PROGRAM general
VAR PERSISTENT
	//System date time function block
	system_date_time : date_time;
	//Daily reset bit, used throughout the program for any resets
	daily_reset : BOOL;
	//Alarm Acknoweldge unlatch timer
	alarm_ack_ton : ton;
	//Alarm Reset unlatch timer
	alarm_reset_ton : ton;
	//Alarm Ack and reset unlatch timer setpoint
	alarm_ack_unlatch_sp : TIME :=T#3S;
	
	safety_reset_ton : TON;
	
	safety_reset AT %Q*  : BOOL;
	safety_error_ack AT %Q* : BOOL;
	safety_run AT %Q*  : BOOL;
	
END_VAR

VAR
	
	safety_reset_ons: R_TRIG;
END_VAR
VAR // added by the converter: edge detectors and wires of the graphical bodies
    _w1 : BOOL;
END_VAR

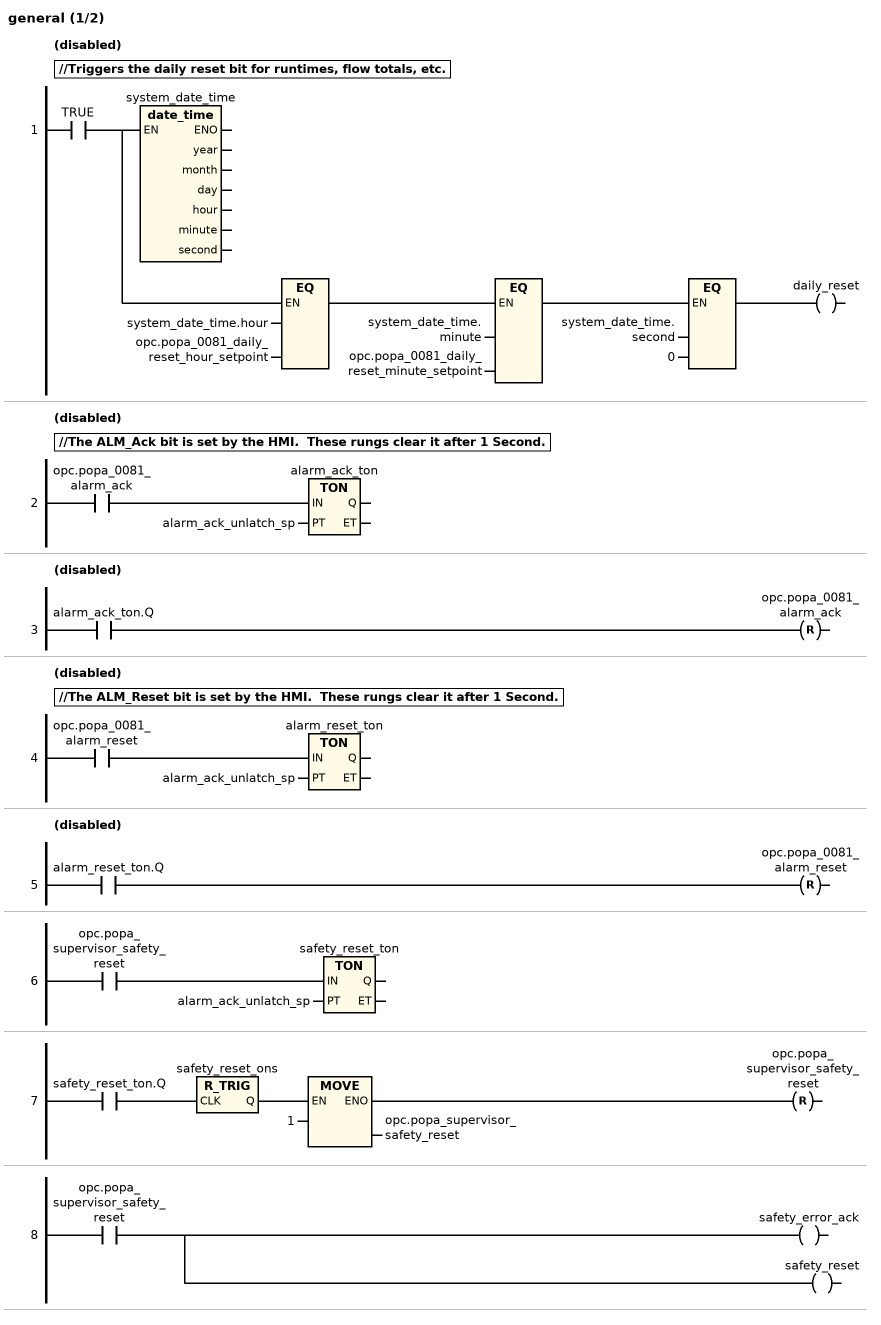
// NETWORK 1 (disabled)
// label: //Triggers the daily reset bit for runtimes, flow totals, etc.
// system_date_time(); // date_time
// daily_reset := system_date_time.hour = opc.popa_0081_daily_reset_hour_setpoint AND system_date_time.minute = opc.popa_0081_daily_reset_minute_setpoint AND system_date_time.second = 0;

// NETWORK 2 (disabled)
// label: //The ALM_Ack bit is set by the HMI.  These rungs clear it after 1 Second.
// alarm_ack_ton(IN := opc.popa_0081_alarm_ack, PT := alarm_ack_unlatch_sp); // TON

// NETWORK 3 (disabled)
// opc.popa_0081_alarm_ack R= alarm_ack_ton.Q;

// NETWORK 4 (disabled)
// label: //The ALM_Reset bit is set by the HMI.  These rungs clear it after 1 Second.
// alarm_reset_ton(IN := opc.popa_0081_alarm_reset, PT := alarm_ack_unlatch_sp); // TON

// NETWORK 5 (disabled)
// opc.popa_0081_alarm_reset R= alarm_reset_ton.Q;

// NETWORK 6
safety_reset_ton(IN := opc.popa_supervisor_safety_reset, PT := alarm_ack_unlatch_sp); // TON

// NETWORK 7
safety_reset_ons(CLK := safety_reset_ton.Q); // R_TRIG
_w1 := safety_reset_ons.Q;
IF _w1 THEN opc.popa_supervisor_safety_reset := 1; END_IF
opc.popa_supervisor_safety_reset R= _w1;

// NETWORK 8
safety_error_ack := opc.popa_supervisor_safety_reset;
safety_reset := opc.popa_supervisor_safety_reset;

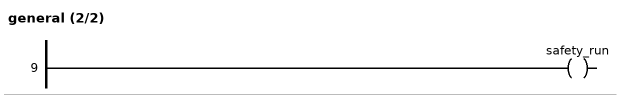
// NETWORK 9
safety_run := TRUE;

END_PROGRAM

(* stored: Version 1.1.0.1, ProductVersion 3.1.4024.15
   POU general: Id {afd5554c-a122-45cd-a612-91df6056dfdf}, SpecialFunc None *)
